// TIA Portal V18 export
DATA_BLOCK "L1_attuatori"   // DB2
{ S7_Optimized_Access := 'TRUE' }
VERSION : 0.1
// stored: AutoNumber true, DBAccessibleFromOPCUA true, DBAccessibleFromWebserver true, IsOnlyStoredInLoadMemory false, IsRetainMemResEnabled false, IsWriteProtectedInAS false, MemoryReserve 100
   VAR RETAIN
      stz_cmd : Array[1.."N_STAZIONI"] of "LGasp_CmdAttuatori";   // N_STAZIONI non inferiore a 20 altrimenti il PC va in errore
   END_VAR
   VAR
      stz_stato : Array[1.."N_STAZIONI"] of "LGasp_StatoAttuatori";   // N_STAZIONI non inferiore a 20 altrimenti il PC va in errore
   END_VAR
BEGIN
END_DATA_BLOCK
